{attribute 'GeneratedUsingTerminal: EJ2914-0000-0017'}
{attribute addProperty BoxType "EJ2914-0000-0017"}
{attribute addProperty Id "FSOEAT %Q*FSOE_1DB604F410"}
{attribute addProperty CRC "3386490621"}
{attribute addProperty Size "10"}
TYPE FSoE_Outputs_C9D9BEFD :
STRUCT
	{attribute addProperty Name "FSOE"}
	FSOE AT %Q* : FSOE_1DB604F4;
END_STRUCT
END_TYPE

(* stored: Version 1.2.0.0, ProductVersion 3.1.4024.9
   DUT FSoE_Outputs_C9D9BEFD: Id {bd90cc6b-9f09-464d-b6c6-9a195bac1734} *)
